(* PLC project Unnamed, Unknown Unnamed 1 *)
(* stored: creationDateTime 2026-03-04T10:29:53, modificationDateTime 2026-03-04T10:29:53 *)

FUNCTION_BLOCK MODBEE_ADD_REGISTER
  VAR_INPUT
    REG : BYTE;
    ADDRESS : WORD;
    VAR_BOOL : BOOL;
    VAR_INT : INT;
  END_VAR
  VAR_OUTPUT
    DONE : BOOL;
    ERROR : BOOL;
  END_VAR
  VAR
    hasBeenInitialized : BOOL := 0;
  END_VAR

            {{
MODBEE_ADD_REGISTER_VARS vars;
vars.REG = &data__->REG.value;
vars.ADDRESS = &data__->ADDRESS.value;
vars.VAR_BOOL = &data__->VAR_BOOL.value;
vars.VAR_INT = &data__->VAR_INT.value;
vars.DONE = &data__->DONE.value;
vars.ERROR = &data__->ERROR.value;
}}
if hasBeenInitialized = False then
{{
modbee_add_register_setup(&vars);
}}
hasBeenInitialized := True;
end_if;
{{
modbee_add_register_loop(&vars);
}}
          
END_FUNCTION_BLOCK

FUNCTION_BLOCK MODBEE_CONFIG
  VAR
    hasBeenInitialized : BOOL := 0;
  END_VAR

            {{
MODBEE_CONFIG_VARS vars;
}}
if hasBeenInitialized = False then
{{
modbee_config_setup(&vars);
}}
hasBeenInitialized := True;
end_if;
{{
modbee_config_loop(&vars);
}}
          
END_FUNCTION_BLOCK

FUNCTION_BLOCK MODBEE_HAT_PWR
  VAR_INPUT
    EN_HAT_POWER : BOOL;
  END_VAR
  VAR
    hasBeenInitialized : BOOL := 0;
  END_VAR

            {{
MODBEE_HAT_PWR_VARS vars;
vars.EN_HAT_POWER = &data__->EN_HAT_POWER.value;
}}
if hasBeenInitialized = False then
{{
modbee_hat_pwr_setup(&vars);
}}
hasBeenInitialized := True;
end_if;
{{
modbee_hat_pwr_loop(&vars);
}}
          
END_FUNCTION_BLOCK

FUNCTION_BLOCK MODBEE_HW_CONFIG
  VAR
    hasBeenInitialized : BOOL := 0;
  END_VAR

            {{
MODBEE_HW_CONFIG_VARS vars;
}}
if hasBeenInitialized = False then
{{
modbee_hw_config_setup(&vars);
}}
hasBeenInitialized := True;
end_if;
{{
modbee_hw_config_loop(&vars);
}}
          
END_FUNCTION_BLOCK

FUNCTION_BLOCK MODBEE_HW_INPUTS
  VAR_OUTPUT
    DX01 : BOOL;
    DX02 : BOOL;
    DX03 : BOOL;
    DX04 : BOOL;
    DX05 : BOOL;
    DX06 : BOOL;
    DX07 : BOOL;
    DX08 : BOOL;
    AX01_Scaled : REAL;
    AX02_Scaled : REAL;
    AX03_Scaled : REAL;
    AX04_Scaled : REAL;
  END_VAR
  VAR
    hasBeenInitialized : BOOL := 0;
  END_VAR

            {{
MODBEE_HW_INPUTS_VARS vars;
vars.DX01 = &data__->DX01.value;
vars.DX02 = &data__->DX02.value;
vars.DX03 = &data__->DX03.value;
vars.DX04 = &data__->DX04.value;
vars.DX05 = &data__->DX05.value;
vars.DX06 = &data__->DX06.value;
vars.DX07 = &data__->DX07.value;
vars.DX08 = &data__->DX08.value;
vars.AX01_SCALED = &data__->AX01_SCALED.value;
vars.AX02_SCALED = &data__->AX02_SCALED.value;
vars.AX03_SCALED = &data__->AX03_SCALED.value;
vars.AX04_SCALED = &data__->AX04_SCALED.value;
}}
if hasBeenInitialized = False then
{{
modbee_hw_inputs_setup(&vars);
}}
hasBeenInitialized := True;
end_if;
{{
modbee_hw_inputs_loop(&vars);
}}
          
END_FUNCTION_BLOCK

FUNCTION_BLOCK MODBEE_HW_OUTPUTS
  VAR_INPUT
    DY01 : BOOL;
    DY02 : BOOL;
    DY03 : BOOL;
    DY04 : BOOL;
    DY05 : BOOL;
    DY06 : BOOL;
    DY07 : BOOL;
    DY08 : BOOL;
    AY01_Scaled : REAL;
    AY02_Scaled : REAL;
  END_VAR
  VAR
    hasBeenInitialized : BOOL := 0;
  END_VAR

            {{
MODBEE_HW_OUTPUTS_VARS vars;
vars.DY01 = &data__->DY01.value;
vars.DY02 = &data__->DY02.value;
vars.DY03 = &data__->DY03.value;
vars.DY04 = &data__->DY04.value;
vars.DY05 = &data__->DY05.value;
vars.DY06 = &data__->DY06.value;
vars.DY07 = &data__->DY07.value;
vars.DY08 = &data__->DY08.value;
vars.AY01_SCALED = &data__->AY01_SCALED.value;
vars.AY02_SCALED = &data__->AY02_SCALED.value;
}}
if hasBeenInitialized = False then
{{
modbee_hw_outputs_setup(&vars);
}}
hasBeenInitialized := True;
end_if;
{{
modbee_hw_outputs_loop(&vars);
}}
          
END_FUNCTION_BLOCK

FUNCTION_BLOCK MODBEE_READ
  VAR_INPUT
    REQ : BOOL;
    NODE_ID : BYTE;
    REG_TYPE : BYTE;
    START_ADDR : WORD;
    LENGTH : BYTE;
  END_VAR
  VAR_OUTPUT
    DONE : BOOL;
    ERROR : BOOL;
    NODE_ONLINE : BOOL;
    COIL_01 : BOOL;
    COIL_02 : BOOL;
    COIL_03 : BOOL;
    COIL_04 : BOOL;
    COIL_05 : BOOL;
    COIL_06 : BOOL;
    COIL_07 : BOOL;
    COIL_08 : BOOL;
    REG_01 : INT;
    REG_02 : INT;
    REG_03 : INT;
    REG_04 : INT;
    REG_05 : INT;
    REG_06 : INT;
    REG_07 : INT;
    REG_08 : INT;
  END_VAR
  VAR
    hasBeenInitialized : BOOL := 0;
  END_VAR

            {{
MODBEE_READ_VARS vars;
vars.REQ = &data__->REQ.value;
vars.NODE_ID = &data__->NODE_ID.value;
vars.REG_TYPE = &data__->REG_TYPE.value;
vars.START_ADDR = &data__->START_ADDR.value;
vars.LENGTH = &data__->LENGTH.value;
vars.DONE = &data__->DONE.value;
vars.ERROR = &data__->ERROR.value;
vars.NODE_ONLINE = &data__->NODE_ONLINE.value;
vars.COIL_01 = &data__->COIL_01.value;
vars.COIL_02 = &data__->COIL_02.value;
vars.COIL_03 = &data__->COIL_03.value;
vars.COIL_04 = &data__->COIL_04.value;
vars.COIL_05 = &data__->COIL_05.value;
vars.COIL_06 = &data__->COIL_06.value;
vars.COIL_07 = &data__->COIL_07.value;
vars.COIL_08 = &data__->COIL_08.value;
vars.REG_01 = &data__->REG_01.value;
vars.REG_02 = &data__->REG_02.value;
vars.REG_03 = &data__->REG_03.value;
vars.REG_04 = &data__->REG_04.value;
vars.REG_05 = &data__->REG_05.value;
vars.REG_06 = &data__->REG_06.value;
vars.REG_07 = &data__->REG_07.value;
vars.REG_08 = &data__->REG_08.value;
}}
if hasBeenInitialized = False then
{{
modbee_read_setup(&vars);
}}
hasBeenInitialized := True;
end_if;
{{
modbee_read_loop(&vars);
}}
          
END_FUNCTION_BLOCK

FUNCTION_BLOCK MODBEE_READ_ARRAY
  VAR_INPUT
    REQ : BOOL;
    NODE_ID : BYTE;
    REG_TYPE : BYTE;
    START_ADDR : WORD;
    LENGTH : BYTE;
  END_VAR
  VAR_OUTPUT
    DONE : BOOL;
    ERROR : BOOL;
    NODE_ONLINE : BOOL;
    COILS : ARRAY[0..31] OF BOOL;
    REGS : ARRAY[0..31] OF INT;
  END_VAR
  VAR
    hasBeenInitialized : BOOL := 0;
  END_VAR

            {{
MODBEE_READ_ARRAY_VARS vars;
IEC_BOOL __flat_COILS[32];
IEC_INT __flat_REGS[32];
for (int __i = 0; __i < 32; __i++) __flat_COILS[__i] = data__->COILS.value.table[__i].value;
for (int __i = 0; __i < 32; __i++) __flat_REGS[__i] = data__->REGS.value.table[__i].value;
vars.REQ = &data__->REQ.value;
vars.NODE_ID = &data__->NODE_ID.value;
vars.REG_TYPE = &data__->REG_TYPE.value;
vars.START_ADDR = &data__->START_ADDR.value;
vars.LENGTH = &data__->LENGTH.value;
vars.DONE = &data__->DONE.value;
vars.ERROR = &data__->ERROR.value;
vars.NODE_ONLINE = &data__->NODE_ONLINE.value;
vars.COILS = __flat_COILS - 0;
vars.REGS = __flat_REGS - 0;
}}
if hasBeenInitialized = False then
{{
modbee_read_array_setup(&vars);
}}
hasBeenInitialized := True;
end_if;
{{
modbee_read_array_loop(&vars);
}}
{{
for (int __i = 0; __i < 32; __i++) data__->COILS.value.table[__i].value = __flat_COILS[__i];
for (int __i = 0; __i < 32; __i++) data__->REGS.value.table[__i].value = __flat_REGS[__i];
}}
          
END_FUNCTION_BLOCK

FUNCTION_BLOCK MODBEE_WRITE
  VAR_INPUT
    REQ : BOOL;
    NODE_ID : BYTE;
    REG_TYPE : BYTE;
    START_ADDR : WORD;
    LENGTH : BYTE;
    COIL_01 : BOOL;
    COIL_02 : BOOL;
    COIL_03 : BOOL;
    COIL_04 : BOOL;
    COIL_05 : BOOL;
    COIL_06 : BOOL;
    COIL_07 : BOOL;
    COIL_08 : BOOL;
    REG_01 : INT;
    REG_02 : INT;
    REG_03 : INT;
    REG_04 : INT;
    REG_05 : INT;
    REG_06 : INT;
    REG_07 : INT;
    REG_08 : INT;
  END_VAR
  VAR_OUTPUT
    DONE : BOOL;
    ERROR : BOOL;
    NODE_ONLINE : BOOL;
  END_VAR
  VAR
    hasBeenInitialized : BOOL := 0;
  END_VAR

            {{
MODBEE_WRITE_VARS vars;
vars.REQ = &data__->REQ.value;
vars.NODE_ID = &data__->NODE_ID.value;
vars.REG_TYPE = &data__->REG_TYPE.value;
vars.START_ADDR = &data__->START_ADDR.value;
vars.LENGTH = &data__->LENGTH.value;
vars.COIL_01 = &data__->COIL_01.value;
vars.COIL_02 = &data__->COIL_02.value;
vars.COIL_03 = &data__->COIL_03.value;
vars.COIL_04 = &data__->COIL_04.value;
vars.COIL_05 = &data__->COIL_05.value;
vars.COIL_06 = &data__->COIL_06.value;
vars.COIL_07 = &data__->COIL_07.value;
vars.COIL_08 = &data__->COIL_08.value;
vars.REG_01 = &data__->REG_01.value;
vars.REG_02 = &data__->REG_02.value;
vars.REG_03 = &data__->REG_03.value;
vars.REG_04 = &data__->REG_04.value;
vars.REG_05 = &data__->REG_05.value;
vars.REG_06 = &data__->REG_06.value;
vars.REG_07 = &data__->REG_07.value;
vars.REG_08 = &data__->REG_08.value;
vars.DONE = &data__->DONE.value;
vars.ERROR = &data__->ERROR.value;
vars.NODE_ONLINE = &data__->NODE_ONLINE.value;
}}
if hasBeenInitialized = False then
{{
modbee_write_setup(&vars);
}}
hasBeenInitialized := True;
end_if;
{{
modbee_write_loop(&vars);
}}
          
END_FUNCTION_BLOCK

FUNCTION_BLOCK MODBEE_WRITE_ARRAY
  VAR_INPUT
    REQ : BOOL;
    NODE_ID : BYTE;
    REG_TYPE : BYTE;
    START_ADDR : WORD;
    LENGTH : BYTE;
    COILS : ARRAY[0..31] OF BOOL;
    REGS : ARRAY[0..31] OF INT;
  END_VAR
  VAR_OUTPUT
    DONE : BOOL;
    ERROR : BOOL;
    NODE_ONLINE : BOOL;
  END_VAR
  VAR
    hasBeenInitialized : BOOL := 0;
  END_VAR

            {{
MODBEE_WRITE_ARRAY_VARS vars;
IEC_BOOL __flat_COILS[32];
IEC_INT __flat_REGS[32];
for (int __i = 0; __i < 32; __i++) __flat_COILS[__i] = data__->COILS.value.table[__i].value;
for (int __i = 0; __i < 32; __i++) __flat_REGS[__i] = data__->REGS.value.table[__i].value;
vars.REQ = &data__->REQ.value;
vars.NODE_ID = &data__->NODE_ID.value;
vars.REG_TYPE = &data__->REG_TYPE.value;
vars.START_ADDR = &data__->START_ADDR.value;
vars.LENGTH = &data__->LENGTH.value;
vars.COILS = __flat_COILS - 0;
vars.REGS = __flat_REGS - 0;
vars.DONE = &data__->DONE.value;
vars.ERROR = &data__->ERROR.value;
vars.NODE_ONLINE = &data__->NODE_ONLINE.value;
}}
if hasBeenInitialized = False then
{{
modbee_write_array_setup(&vars);
}}
hasBeenInitialized := True;
end_if;
{{
modbee_write_array_loop(&vars);
}}
          
END_FUNCTION_BLOCK

FUNCTION_BLOCK MODBUS_ADD_REGISTER
  VAR_INPUT
    REG : BYTE;
    ADDRESS : WORD;
    VAR_BOOL : BOOL;
    VAR_INT : INT;
  END_VAR
  VAR_OUTPUT
    DONE : BOOL;
    ERROR : BOOL;
  END_VAR
  VAR
    hasBeenInitialized : BOOL := 0;
  END_VAR

            {{
MODBUS_ADD_REGISTER_VARS vars;
vars.REG = &data__->REG.value;
vars.ADDRESS = &data__->ADDRESS.value;
vars.VAR_BOOL = &data__->VAR_BOOL.value;
vars.VAR_INT = &data__->VAR_INT.value;
vars.DONE = &data__->DONE.value;
vars.ERROR = &data__->ERROR.value;
}}
if hasBeenInitialized = False then
{{
modbus_add_register_setup(&vars);
}}
hasBeenInitialized := True;
end_if;
{{
modbus_add_register_loop(&vars);
}}
          
END_FUNCTION_BLOCK

FUNCTION_BLOCK MODBUS_READ
  VAR_INPUT
    REQ : BOOL;
    SLAVE_ID : BYTE;
    REG_TYPE : BYTE;
    START_ADDR : WORD;
    LENGTH : BYTE;
  END_VAR
  VAR_OUTPUT
    DONE : BOOL;
    ERROR : BOOL;
    COIL_01 : BOOL;
    COIL_02 : BOOL;
    COIL_03 : BOOL;
    COIL_04 : BOOL;
    COIL_05 : BOOL;
    COIL_06 : BOOL;
    COIL_07 : BOOL;
    COIL_08 : BOOL;
    REG_01 : INT;
    REG_02 : INT;
    REG_03 : INT;
    REG_04 : INT;
    REG_05 : INT;
    REG_06 : INT;
    REG_07 : INT;
    REG_08 : INT;
  END_VAR
  VAR
    hasBeenInitialized : BOOL := 0;
  END_VAR

            {{
MODBUS_READ_VARS vars;
vars.REQ = &data__->REQ.value;
vars.SLAVE_ID = &data__->SLAVE_ID.value;
vars.REG_TYPE = &data__->REG_TYPE.value;
vars.START_ADDR = &data__->START_ADDR.value;
vars.LENGTH = &data__->LENGTH.value;
vars.DONE = &data__->DONE.value;
vars.ERROR = &data__->ERROR.value;
vars.COIL_01 = &data__->COIL_01.value;
vars.COIL_02 = &data__->COIL_02.value;
vars.COIL_03 = &data__->COIL_03.value;
vars.COIL_04 = &data__->COIL_04.value;
vars.COIL_05 = &data__->COIL_05.value;
vars.COIL_06 = &data__->COIL_06.value;
vars.COIL_07 = &data__->COIL_07.value;
vars.COIL_08 = &data__->COIL_08.value;
vars.REG_01 = &data__->REG_01.value;
vars.REG_02 = &data__->REG_02.value;
vars.REG_03 = &data__->REG_03.value;
vars.REG_04 = &data__->REG_04.value;
vars.REG_05 = &data__->REG_05.value;
vars.REG_06 = &data__->REG_06.value;
vars.REG_07 = &data__->REG_07.value;
vars.REG_08 = &data__->REG_08.value;
}}
if hasBeenInitialized = False then
{{
modbus_read_setup(&vars);
}}
hasBeenInitialized := True;
end_if;
{{
modbus_read_loop(&vars);
}}
          
END_FUNCTION_BLOCK

FUNCTION_BLOCK MODBUS_READ_ARRAY
  VAR_INPUT
    REQ : BOOL;
    SLAVE_ID : BYTE;
    REG_TYPE : BYTE;
    START_ADDR : WORD;
    LENGTH : BYTE;
  END_VAR
  VAR_OUTPUT
    DONE : BOOL;
    ERROR : BOOL;
    COILS : ARRAY[0..31] OF BOOL;
    REGS : ARRAY[0..31] OF INT;
  END_VAR
  VAR
    hasBeenInitialized : BOOL := 0;
  END_VAR

            {{
MODBUS_READ_ARRAY_VARS vars;
IEC_BOOL __flat_COILS[32];
IEC_INT __flat_REGS[32];
for (int __i = 0; __i < 32; __i++) __flat_COILS[__i] = data__->COILS.value.table[__i].value;
for (int __i = 0; __i < 32; __i++) __flat_REGS[__i] = data__->REGS.value.table[__i].value;
vars.REQ = &data__->REQ.value;
vars.SLAVE_ID = &data__->SLAVE_ID.value;
vars.REG_TYPE = &data__->REG_TYPE.value;
vars.START_ADDR = &data__->START_ADDR.value;
vars.LENGTH = &data__->LENGTH.value;
vars.DONE = &data__->DONE.value;
vars.ERROR = &data__->ERROR.value;
vars.COILS = __flat_COILS - 0;
vars.REGS = __flat_REGS - 0;
}}
if hasBeenInitialized = False then
{{
modbus_read_array_setup(&vars);
}}
hasBeenInitialized := True;
end_if;
{{
modbus_read_array_loop(&vars);
}}
{{
for (int __i = 0; __i < 32; __i++) data__->COILS.value.table[__i].value = __flat_COILS[__i];
for (int __i = 0; __i < 32; __i++) data__->REGS.value.table[__i].value = __flat_REGS[__i];
}}
          
END_FUNCTION_BLOCK

FUNCTION_BLOCK MODBUS_WRITE
  VAR_INPUT
    REQ : BOOL;
    SLAVE_ID : BYTE;
    REG_TYPE : BYTE;
    START_ADDR : WORD;
    LENGTH : BYTE;
    COIL_01 : BOOL;
    COIL_02 : BOOL;
    COIL_03 : BOOL;
    COIL_04 : BOOL;
    COIL_05 : BOOL;
    COIL_06 : BOOL;
    COIL_07 : BOOL;
    COIL_08 : BOOL;
    REG_01 : INT;
    REG_02 : INT;
    REG_03 : INT;
    REG_04 : INT;
    REG_05 : INT;
    REG_06 : INT;
    REG_07 : INT;
    REG_08 : INT;
  END_VAR
  VAR_OUTPUT
    DONE : BOOL;
    ERROR : BOOL;
  END_VAR
  VAR
    hasBeenInitialized : BOOL := 0;
  END_VAR

            {{
MODBUS_WRITE_VARS vars;
vars.REQ = &data__->REQ.value;
vars.SLAVE_ID = &data__->SLAVE_ID.value;
vars.REG_TYPE = &data__->REG_TYPE.value;
vars.START_ADDR = &data__->START_ADDR.value;
vars.LENGTH = &data__->LENGTH.value;
vars.COIL_01 = &data__->COIL_01.value;
vars.COIL_02 = &data__->COIL_02.value;
vars.COIL_03 = &data__->COIL_03.value;
vars.COIL_04 = &data__->COIL_04.value;
vars.COIL_05 = &data__->COIL_05.value;
vars.COIL_06 = &data__->COIL_06.value;
vars.COIL_07 = &data__->COIL_07.value;
vars.COIL_08 = &data__->COIL_08.value;
vars.REG_01 = &data__->REG_01.value;
vars.REG_02 = &data__->REG_02.value;
vars.REG_03 = &data__->REG_03.value;
vars.REG_04 = &data__->REG_04.value;
vars.REG_05 = &data__->REG_05.value;
vars.REG_06 = &data__->REG_06.value;
vars.REG_07 = &data__->REG_07.value;
vars.REG_08 = &data__->REG_08.value;
vars.DONE = &data__->DONE.value;
vars.ERROR = &data__->ERROR.value;
}}
if hasBeenInitialized = False then
{{
modbus_write_setup(&vars);
}}
hasBeenInitialized := True;
end_if;
{{
modbus_write_loop(&vars);
}}
          
END_FUNCTION_BLOCK

FUNCTION_BLOCK MODBUS_WRITE_ARRAY
  VAR_INPUT
    REQ : BOOL;
    SLAVE_ID : BYTE;
    REG_TYPE : BYTE;
    START_ADDR : WORD;
    LENGTH : BYTE;
    COILS : ARRAY[0..31] OF BOOL;
    REGS : ARRAY[0..31] OF INT;
  END_VAR
  VAR_OUTPUT
    DONE : BOOL;
    ERROR : BOOL;
  END_VAR
  VAR
    hasBeenInitialized : BOOL := 0;
  END_VAR

            {{
MODBUS_WRITE_ARRAY_VARS vars;
IEC_BOOL __flat_COILS[32];
IEC_INT __flat_REGS[32];
for (int __i = 0; __i < 32; __i++) __flat_COILS[__i] = data__->COILS.value.table[__i].value;
for (int __i = 0; __i < 32; __i++) __flat_REGS[__i] = data__->REGS.value.table[__i].value;
vars.REQ = &data__->REQ.value;
vars.SLAVE_ID = &data__->SLAVE_ID.value;
vars.REG_TYPE = &data__->REG_TYPE.value;
vars.START_ADDR = &data__->START_ADDR.value;
vars.LENGTH = &data__->LENGTH.value;
vars.COILS = __flat_COILS - 0;
vars.REGS = __flat_REGS - 0;
vars.DONE = &data__->DONE.value;
vars.ERROR = &data__->ERROR.value;
}}
if hasBeenInitialized = False then
{{
modbus_write_array_setup(&vars);
}}
hasBeenInitialized := True;
end_if;
{{
modbus_write_array_loop(&vars);
}}
          
END_FUNCTION_BLOCK

PROGRAM main
  VAR
    MODBEE_HW_INPUTS0 : MODBEE_HW_INPUTS;
    MODBEE_HW_OUTPUTS0 : MODBEE_HW_OUTPUTS;
    start : BOOL;
    stop : BOOL;
    run : BOOL;
    MODBUS_WRITE0 : MODBUS_WRITE;
    MB_SLAVE_DO01 : BOOL;
    MB_SLAVE_DO02 : BOOL;
    MB_SLAVE_DO03 : BOOL;
    MB_SLAVE_DO04 : BOOL;
    MB_SLAVE_DO05 : BOOL;
    MB_SLAVE_DO06 : BOOL;
    MB_SLAVE_DO07 : BOOL;
    MB_SLAVE_DO08 : BOOL;
    MODBUS_READ0 : MODBUS_READ;
    MB_SLAVE_DI01 : BOOL;
    MB_SLAVE_DI02 : BOOL;
    MB_SLAVE_DI03 : BOOL;
    MB_SLAVE_DI05 : BOOL;
    MB_SLAVE_DI04 : BOOL;
    MB_SLAVE_DI06 : BOOL;
    MB_SLAVE_DI07 : BOOL;
    MB_SLAVE_DI08 : BOOL;
    MB_WRITE_COILS_DONE : BOOL;
    MB_READ_COILS_DONE : BOOL;
    TON0 : TON;
    TON1 : TON;
    TON1_DONE : BOOL;
    TON0_DONE : BOOL;
    MODBUS_READ1 : MODBUS_READ;
    MB_READ_REGS_DONE : BOOL;
    MB_SLAVE_AI01 : INT;
    MB_SLAVE_AI02 : INT;
    MB_SLAVE_AI03 : INT;
    MB_SLAVE_AI04 : INT;
    MODBUS_WRITE1 : MODBUS_WRITE;
    MB_WRITE_REGS_DONE : BOOL;
    MB_SLAVE_AO01 : REAL;
    MB_SLAVE_AO02 : REAL;
    MB_SLAVE_AO03 : REAL;
    MB_SLAVE_AO04 : REAL;
    MB_SLAVE_AO5 : INT;
    MB_SLAVE_AO01_TEMP : INT;
    MB_SLAVE_AO02_TEMP : INT;
    MB_WRITE_REGS_DONE0 : BOOL;
  END_VAR

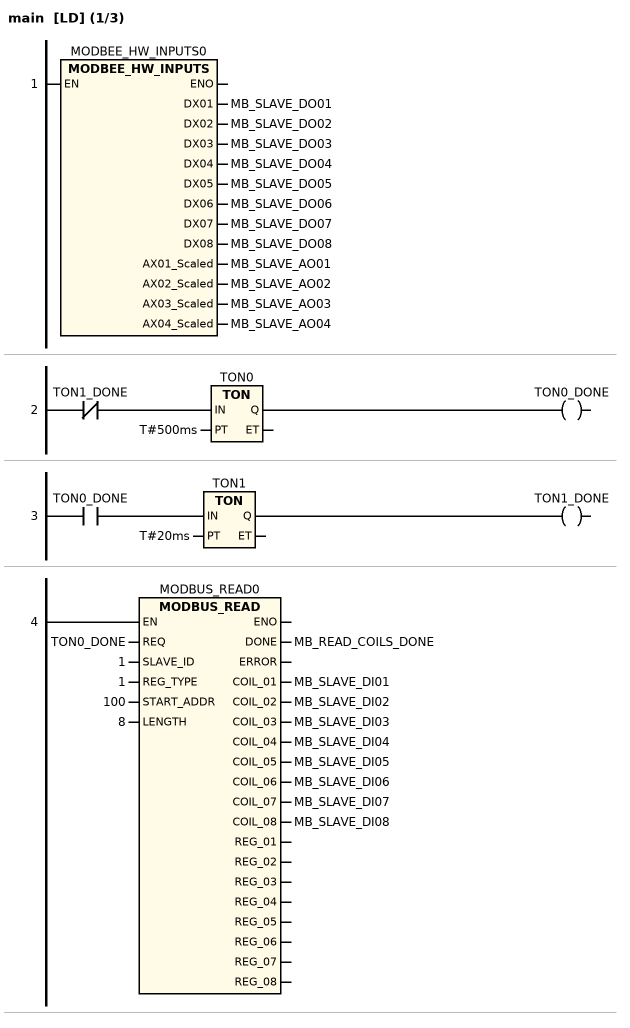
(* LD diagram, written out as Structured Text *)
TON0(IN := NOT TON1_DONE, PT := T#500ms);
TON0_DONE := TON0.Q;
TON1(IN := TON0_DONE, PT := T#20ms);
TON1_DONE := TON1.Q;
MODBEE_HW_INPUTS0();
MB_SLAVE_DO01 := MODBEE_HW_INPUTS0.DX01;
MB_SLAVE_DO02 := MODBEE_HW_INPUTS0.DX02;
MB_SLAVE_DO03 := MODBEE_HW_INPUTS0.DX03;
MB_SLAVE_DO04 := MODBEE_HW_INPUTS0.DX04;
MB_SLAVE_DO05 := MODBEE_HW_INPUTS0.DX05;
MB_SLAVE_DO06 := MODBEE_HW_INPUTS0.DX06;
MB_SLAVE_DO07 := MODBEE_HW_INPUTS0.DX07;
MB_SLAVE_DO08 := MODBEE_HW_INPUTS0.DX08;
MB_SLAVE_AO01 := MODBEE_HW_INPUTS0.AX01_Scaled;
MB_SLAVE_AO02 := MODBEE_HW_INPUTS0.AX02_Scaled;
MB_SLAVE_AO03 := MODBEE_HW_INPUTS0.AX03_Scaled;
MB_SLAVE_AO04 := MODBEE_HW_INPUTS0.AX04_Scaled;
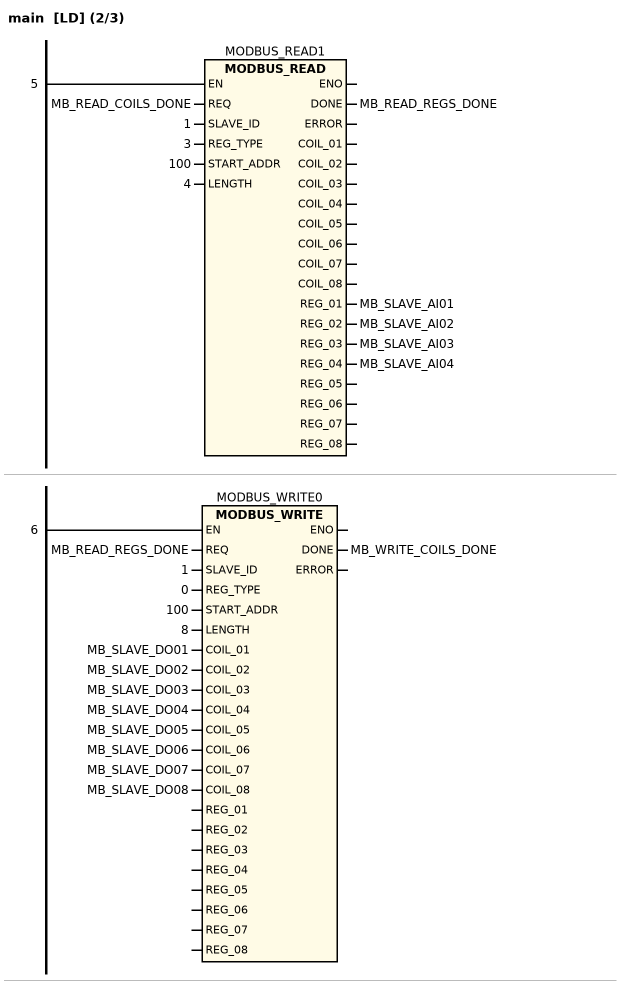
MODBUS_READ0(REQ := TON0_DONE, SLAVE_ID := 1, REG_TYPE := 1, START_ADDR := 100, LENGTH := 8);
MB_READ_COILS_DONE := MODBUS_READ0.DONE;
MB_SLAVE_DI01 := MODBUS_READ0.COIL_01;
MB_SLAVE_DI02 := MODBUS_READ0.COIL_02;
MB_SLAVE_DI03 := MODBUS_READ0.COIL_03;
MB_SLAVE_DI04 := MODBUS_READ0.COIL_04;
MB_SLAVE_DI05 := MODBUS_READ0.COIL_05;
MB_SLAVE_DI06 := MODBUS_READ0.COIL_06;
MB_SLAVE_DI07 := MODBUS_READ0.COIL_07;
MB_SLAVE_DI08 := MODBUS_READ0.COIL_08;
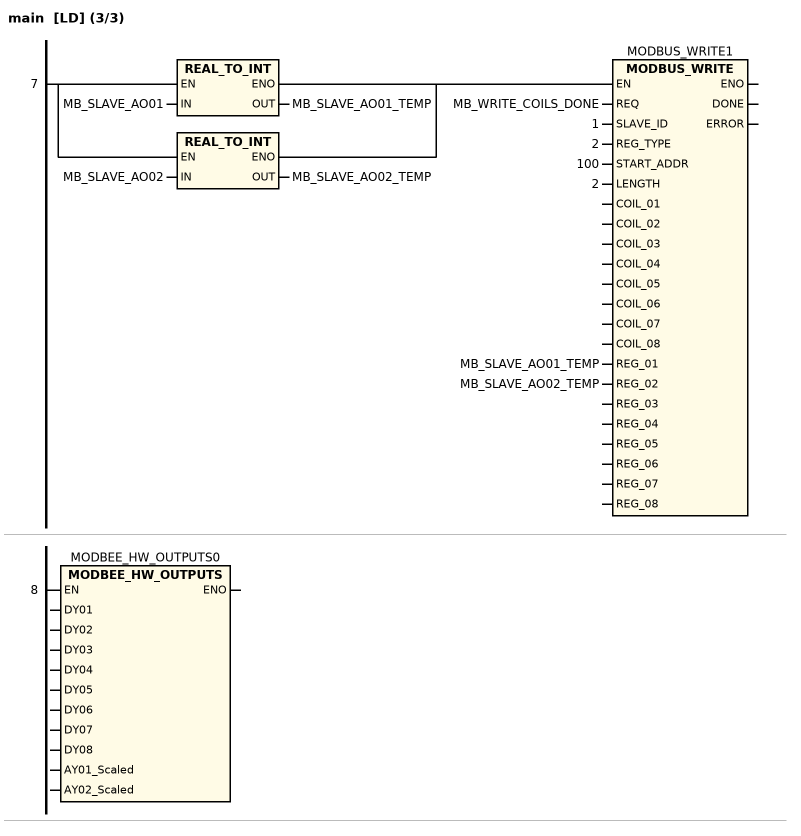
MODBUS_READ1(REQ := MB_READ_COILS_DONE, SLAVE_ID := 1, REG_TYPE := 3, START_ADDR := 100, LENGTH := 4);
MB_READ_REGS_DONE := MODBUS_READ1.DONE;
MB_SLAVE_AI01 := MODBUS_READ1.REG_01;
MB_SLAVE_AI02 := MODBUS_READ1.REG_02;
MB_SLAVE_AI03 := MODBUS_READ1.REG_03;
MB_SLAVE_AI04 := MODBUS_READ1.REG_04;
MODBUS_WRITE0(REQ := MB_READ_REGS_DONE, SLAVE_ID := 1, REG_TYPE := 0, START_ADDR := 100, LENGTH := 8, COIL_01 := MB_SLAVE_DO01, COIL_02 := MB_SLAVE_DO02, COIL_03 := MB_SLAVE_DO03, COIL_04 := MB_SLAVE_DO04, COIL_05 := MB_SLAVE_DO05, COIL_06 := MB_SLAVE_DO06, COIL_07 := MB_SLAVE_DO07, COIL_08 := MB_SLAVE_DO08);
MB_WRITE_COILS_DONE := MODBUS_WRITE0.DONE;
MB_SLAVE_AO01_TEMP := REAL_TO_INT(MB_SLAVE_AO01);
MB_SLAVE_AO02_TEMP := REAL_TO_INT(MB_SLAVE_AO02);
MODBUS_WRITE1(REQ := MB_WRITE_COILS_DONE, SLAVE_ID := 1, REG_TYPE := 2, START_ADDR := 100, LENGTH := 2, REG_01 := MB_SLAVE_AO01_TEMP, REG_02 := MB_SLAVE_AO02_TEMP);
MODBEE_HW_OUTPUTS0();
END_PROGRAM

PROGRAM modbee
  VAR
    MODBEE_HW_CONFIG0 : MODBEE_HW_CONFIG;
  END_VAR

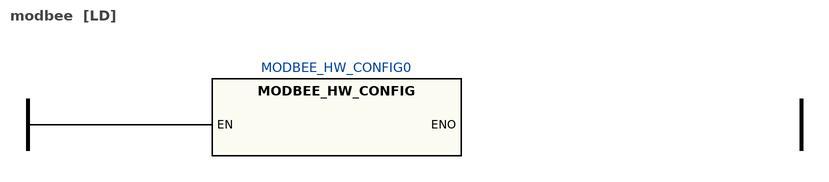
(* LD diagram, written out as Structured Text *)
MODBEE_HW_CONFIG0();
END_PROGRAM

CONFIGURATION Config0
  RESOURCE Res0 ON PLC
    TASK task0(INTERVAL := T#10ms, PRIORITY := 1);
    TASK Task1(INTERVAL := T#1ms, PRIORITY := 0);
    PROGRAM instance0 WITH task0 : main;
    PROGRAM instance1 WITH Task1 : modbee;
  END_RESOURCE
END_CONFIGURATION
